Universal Robots PolyScope program: cottonMotorOff.urp

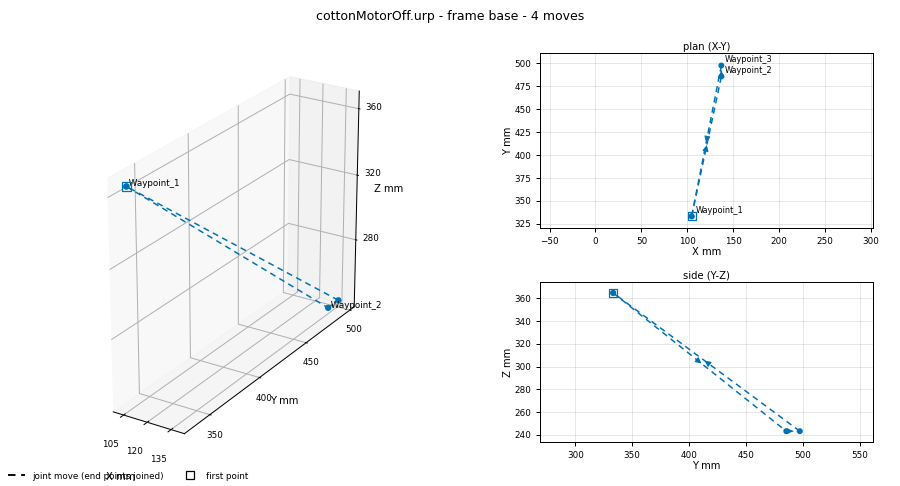
[picture p0: tool path of cottonMotorOff.urp in frame base, 4 of 6 moves have a stored position in this frame; points joined in program order, loops and branches not executed]
Program cottonMotorOff (installation=default directory=/programs/DavidMelin createdIn=5.12.4.1101661 lastSavedIn=5.12.4.1101661 robotSerialNumber=20225502378)
Calibrated DH parameters: a=[0.00022, -0.425328, -0.389701, 0.000059, 0.000065, 0]; d=[0.162608, 0.803456, 9.992211, -10.662202, 0.099702, 0.099559]; alpha=[1.570756, 0.001543, 0.004316, 1.570651, -1.570122, 0]; deltaTheta=[0, 0.002917, 0.116094, -0.119008, 0, -0.000001]
Robot Program (runOnlyOnce=true)
  MoveJ speed 60 deg/s, acceleration 80 deg/s^2 (useActiveTCP=true) feature=Base
    Waypoint Waypoint (Variable): variable=cotonHomePos
  URCap Gripper (Robotiq_Grippers, Robotiq Inc.) dataModel(position=100.0, force=0.0, speed=100.0, positionInDouble=100.0, forceInDouble=0.0, speedInDouble=100.0, slaveIds=[9], blocking=true)
  MoveJ speed 60 deg/s, acceleration 80 deg/s^2 (useActiveTCP=true) feature=Base
    Waypoint Waypoint_1: TCP in base x=104.638 y=333.285 z=364.778 mm, rx=-2.4906 ry=0.0957 rz=-0.1131 rad; joints [98.538, -64.729, -139.703, -29.68, 79.086, 9.451] deg
    Waypoint Waypoint_2: TCP in base x=137 y=485.518 z=243.196 mm, rx=-2.395 ry=0.1184 rz=-0.0957 rad; joints [90.955, -106.171, -129.043, 7.481, 83.548, 4.286] deg
    Waypoint Waypoint_3: TCP in base x=136.97 y=497.445 z=243.204 mm, rx=-2.395 ry=0.1183 rz=-0.0957 rad; joints [90.933, -107.352, -127.222, 6.845, 83.569, 4.269] deg
    Waypoint Waypoint_4: TCP in base x=104.65 y=333.289 z=364.771 mm, rx=-2.4906 ry=0.0958 rz=-0.1131 rad; joints [98.536, -64.731, -139.702, -29.679, 79.086, 9.452] deg
    Waypoint Waypoint (Variable): variable=cotonHomePos
